TYPE ST_DALIBridgeInputEvent :
STRUCT
	parameters : ST_DALIBridgeInputEventParams;
	error      : BOOL;
	status     : UDINT;
	message    : STRING(255);
	data       : WORD;
END_STRUCT
END_TYPE

(* stored: Version 1.1.0.1, ProductVersion 3.1.4024.10
   DUT ST_DALIBridgeInputEvent: Id {f5264ecb-13d8-4782-b9fa-850cc5c69f2a} *)
